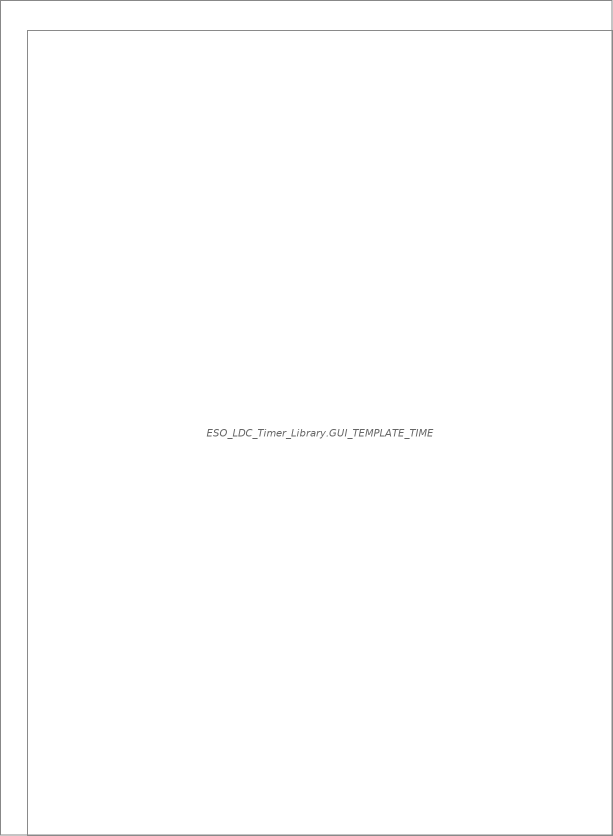
VISUALIZATION GUI_TIMER  // 613x836
    Frame (27,30 586x806)
        shows ESO_LDC_Timer_Library.GUI_TEMPLATE_TIME(m_Instance := MAIN.fbTimer)
END_VISUALIZATION

(* stored: Version 1.1.0.1, ProductVersion 3.1.4024.9
   Visu GUI_TIMER: Id {3f7806fa-abf6-477e-b606-fdc040fa89c4} *)
